FUNCTION_BLOCK RunGroupNode EXTENDS RunUnitGeneric
VAR_INPUT
	members : ARRAY[0..7] OF POINTER TO RunUnitGeneric;
END_VAR
VAR
	nCounter : DINT;
END_VAR

SUPER^();

CASE outputState OF 
	//------------Initialize
	eSpecialStates.INITIAL_STATE_1:
		// group node start initializing
		bSerialTransition := TRUE;
		
		//scan if all initialized
		FOR nCounter := 0 TO 7 DO
			IF members[nCounter] <> 0 THEN
				bSerialTransition := bSerialTransition AND members[nCounter]^.Initialize();
			END_IF		
		END_FOR
		
		// wait upper to inform starting
		IF bSerialTransition THEN
			NextState:=eSpecialStates.INITIAL_END;
		END_IF

	eSpecialStates.GENERIC_GROUP_START:
		//then wait command to trigger all station into working state
		FOR nCounter := 0 TO 7 DO
			IF members[nCounter] <> 0 THEN
				members[nCounter]^.NextState := eSpecialStates.GENERIC_GROUP_START;
			END_IF
		END_FOR
		bSerialTransition := TRUE; //group idle
END_CASE

METHOD FB_init : BOOL
VAR_INPUT
	bInitRetains : BOOL; // if TRUE, the retain variables are initialized (warm start / cold start)
	bInCopyCode : BOOL;  // if TRUE, the instance afterwards gets moved into the copy code (online change)
	
	argParent : POINTER TO RunUnitGeneric;
	argSlotBase : POINTER TO RunMaterial;
	argSlotLast : POINTER TO RunMaterial;
END_VAR
//initialize 
Parent := argParent;
SlotBase := argSlotBase;
SlotLast := argSlotLast;
//
IF bInitRetains THEN
	NextState := eSpecialStates.INITIAL_BEGIN;
END_IF
END_METHOD

METHOD Initialize : BOOL
VAR_INPUT
END_VAR
VAR
	nCounter : int;
END_VAR
//once initializing method call , redirect current state to initalizing region
IF (TO_UINT(State) AND TO_UINT(eSpecialStates.INITIAL_REGION)) =0 THEN
	NextState := eSpecialStates.INITIAL_BEGIN; //not in intializing region , change
END_IF

Initialize := (State = eSpecialStates.INITIAL_END);

IF Initialize THEN
	//clear all remained signal
	FOR nCounter:=1 TO 32 BY 1 DO
		slaveWorkingSignal[nCounter] := FALSE;
	END_FOR
	//clear all internal status
	bEnStep := FALSE;
	bTrigStep := FALSE;
	bIsBypassed := FALSE;
	bWorkingOverride := FALSE;
	bMaterialOverride := FALSE;	
END_IF
END_METHOD

END_FUNCTION_BLOCK

(* stored: Version 1.1.0.1, ProductVersion 3.1.4024.0
   POU RunGroupNode: Id {b9fe6715-7af9-4baf-8aa9-637788ac271f}, SpecialFunc None
   Method FB_init: Id {065bd92a-f7f5-4f57-987a-22d42058151c}
   Method Initialize: Id {eb434dc7-b60c-4ac2-84bb-e6d7d85262c7} *)
